{attribute 'qualified_only'}
VAR_GLOBAL
	fbCrititcalSection : FB_IecCriticalSection;
	fbDoWork		   : FB_DoWork;
END_VAR

(* stored: Version 1.1.0.1, ProductVersion 3.1.4026.18
   GVL GVL: Id {19cfac5f-7d6b-4a04-8d11-affb2848f9ce} *)
